(* IEC 61131-3 sources: Lasal/CPU_5344_V01/Class/MillPlane, 1 file *)

(* ---- MillPlane.st ---- *)
(*!
<Class
	Name               = "MillPlane"
	Revision           = "0.0"
	RealtimeTask       = "false"
	CyclicTask         = "false"
	BackgroundTask     = "false"
	Sigmatek           = "false"
	OSInterface        = "false"
	HighPriority       = "false"
	Automatic          = "false"
	UpdateMode         = "Prescan"
	SharedCommandTable = "true"
	Objectsize         = "(390,360)">
	<Channels>
		<Server Name="amount" Visualized="true" Initialize="false" WriteProtected="false" Retentive="false"/>
		<Server Name="ClassSvr" Visualized="false" Initialize="false" WriteProtected="true" Retentive="false"/>
		<Server Name="depth" Visualized="true" Initialize="false" WriteProtected="false" Retentive="false"/>
		<Server Name="feedRate" Visualized="true" Initialize="false" WriteProtected="false" Retentive="false"/>
		<Server Name="firsIdx" Visualized="true" Initialize="false" WriteProtected="false" Retentive="false"/>
		<Server Name="lowerRate" Visualized="true" Initialize="false" WriteProtected="false" Retentive="false"/>
		<Server Name="rnr" Visualized="true" Initialize="false" WriteProtected="false" Retentive="false"/>
		<Client Name="line1" Required="true" Internal="true"/>
		<Client Name="line2" Required="true" Internal="true"/>
		<Client Name="line3" Required="true" Internal="true"/>
		<Client Name="line4" Required="true" Internal="true"/>
		<Client Name="line5" Required="true" Internal="true"/>
		<Client Name="line6" Required="true" Internal="true"/>
	</Channels>
	<Network Name="MillPlane">
		<!-- List of Components in this network -->
		<Components>
			<Object
				Name       = "line1"
				Class      = "MillLine"
				Position   = "(150,120)"
				Visualized = "true">
				<Channels>
					<Server Name="ClassSvr"/>
					<Server Name="middleX"/>
					<Server Name="middleY"/>
					<Server Name="millType"/>
					<Server Name="radius"/>
					<Server Name="rnr"/>
					<Server Name="xGoal"/>
					<Server Name="yGoal"/>
				</Channels>
			</Object>
			<Object
				Name       = "line2"
				Class      = "MillLine"
				Position   = "(150,690)"
				Visualized = "true">
				<Channels>
					<Server Name="ClassSvr"/>
					<Server Name="middleX"/>
					<Server Name="middleY"/>
					<Server Name="millType"/>
					<Server Name="radius"/>
					<Server Name="rnr"/>
					<Server Name="xGoal"/>
					<Server Name="yGoal"/>
				</Channels>
			</Object>
			<Object
				Name       = "line3"
				Class      = "MillLine"
				Position   = "(720,120)"
				Visualized = "true">
				<Channels>
					<Server Name="ClassSvr"/>
					<Server Name="middleX"/>
					<Server Name="middleY"/>
					<Server Name="millType"/>
					<Server Name="radius"/>
					<Server Name="rnr"/>
					<Server Name="xGoal"/>
					<Server Name="yGoal"/>
				</Channels>
			</Object>
			<Object
				Name       = "line4"
				Class      = "MillLine"
				Position   = "(720,690)"
				Visualized = "true">
				<Channels>
					<Server Name="ClassSvr"/>
					<Server Name="middleX"/>
					<Server Name="middleY"/>
					<Server Name="millType"/>
					<Server Name="radius"/>
					<Server Name="rnr"/>
					<Server Name="xGoal"/>
					<Server Name="yGoal"/>
				</Channels>
			</Object>
			<Object
				Name       = "line5"
				Class      = "MillLine"
				Position   = "(1260,120)"
				Visualized = "true">
				<Channels>
					<Server Name="ClassSvr"/>
					<Server Name="middleX"/>
					<Server Name="middleY"/>
					<Server Name="millType"/>
					<Server Name="radius"/>
					<Server Name="rnr"/>
					<Server Name="xGoal"/>
					<Server Name="yGoal"/>
				</Channels>
			</Object>
			<Object
				Name       = "line6"
				Class      = "MillLine"
				Position   = "(1260,690)"
				Visualized = "true">
				<Channels>
					<Server Name="ClassSvr"/>
					<Server Name="middleX"/>
					<Server Name="middleY"/>
					<Server Name="millType"/>
					<Server Name="radius"/>
					<Server Name="rnr"/>
					<Server Name="xGoal"/>
					<Server Name="yGoal"/>
				</Channels>
			</Object>
		</Components>
		<Comments>
		</Comments>
		<!-- List of Connections in this network -->
		<Connections>
			<Connection Source="this.line1" Destination="line1.ClassSvr"/>
			<Connection Source="this.line2" Destination="line2.ClassSvr"/>
			<Connection Source="this.line4" Destination="line4.ClassSvr"/>
			<Connection Source="this.line3" Destination="line3.ClassSvr"/>
			<Connection Source="this.line5" Destination="line5.ClassSvr"/>
			<Connection Source="this.line6" Destination="line6.ClassSvr"/>
		</Connections>
		<!-- Headerfiles -->
		<Options>
		</Options>
	</Network>
</Class>
*)
MillPlane : CLASS
  //Servers:
	ClassSvr 	: SvrChCmd_DINT;
	rnr 	: SvrCh_DINT;
	depth 	: SvrCh_DINT;
	amount 	: SvrCh_DINT;
	feedRate 	: SvrCh_DINT;
	lowerRate 	: SvrCh_DINT;
	firsIdx 	: SvrCh_DINT;
  //Clients:
	line1 	: CltChCmd_MillLine;
	line2 	: CltChCmd_MillLine;
	line3 	: CltChCmd_MillLine;
	line4 	: CltChCmd_MillLine;
	line5 	: CltChCmd_MillLine;
	line6 	: CltChCmd_MillLine;
  //Variables:
		ptr 	: ^strMillPlane;
  //Functions:

	FUNCTION GLOBAL WritePtr
		VAR_INPUT
			iPtr 	: ^strMillPlane;
		END_VAR;

	FUNCTION WriteServers;

	FUNCTION VIRTUAL GLOBAL depth::Write
		VAR_INPUT
			input (EAX) 	: DINT;
		END_VAR
		VAR_OUTPUT
			result (EAX) 	: DINT;
		END_VAR;

	FUNCTION VIRTUAL GLOBAL amount::Write
		VAR_INPUT
			input (EAX) 	: DINT;
		END_VAR
		VAR_OUTPUT
			result (EAX) 	: DINT;
		END_VAR;

	FUNCTION VIRTUAL GLOBAL feedRate::Write
		VAR_INPUT
			input (EAX) 	: DINT;
		END_VAR
		VAR_OUTPUT
			result (EAX) 	: DINT;
		END_VAR;

	FUNCTION VIRTUAL GLOBAL lowerRate::Write
		VAR_INPUT
			input (EAX) 	: DINT;
		END_VAR
		VAR_OUTPUT
			result (EAX) 	: DINT;
		END_VAR;

	FUNCTION VIRTUAL GLOBAL firsIdx::Write
		VAR_INPUT
			input (EAX) 	: DINT;
		END_VAR
		VAR_OUTPUT
			result (EAX) 	: DINT;
		END_VAR;
  //Tables:
	FUNCTION @STD
		VAR_OUTPUT
			ret_code	: CONFSTATES;
		END_VAR;
	FUNCTION GLOBAL TAB @CT_;
END_CLASS;

#pragma using MillLine

FUNCTION VIRTUAL GLOBAL MillPlane::depth::Write
	VAR_INPUT
		input (EAX) 	: DINT;
	END_VAR
	VAR_OUTPUT
		result (EAX) 	: DINT;
	END_VAR

  if ptr <> NIL then
    depth := input;
    ptr^.depth := depth;
    result := depth;
  else
    result := ACCESS_DENIED;
  end_if;

END_FUNCTION

FUNCTION VIRTUAL GLOBAL MillPlane::amount::Write
	VAR_INPUT
		input (EAX) 	: DINT;
	END_VAR
	VAR_OUTPUT
		result (EAX) 	: DINT;
	END_VAR

  if ptr <> NIL then
    amount := input;
    ptr^.amount := amount;
    result := amount;
  else
    result := ACCESS_DENIED;
  end_if;

END_FUNCTION

FUNCTION VIRTUAL GLOBAL MillPlane::feedRate::Write
	VAR_INPUT
		input (EAX) 	: DINT;
	END_VAR
	VAR_OUTPUT
		result (EAX) 	: DINT;
	END_VAR

  if ptr <> NIL then
    feedRate := input;
    ptr^.feedRate := feedRate;
    result := feedRate;
  else
    result := ACCESS_DENIED;
  end_if;

END_FUNCTION

FUNCTION GLOBAL MillPlane::WritePtr
	VAR_INPUT
		iPtr 	: ^strMillPlane;
	END_VAR

  ptr := iPtr;
  WriteServers();
  firsIdx.Write(input:=0);

END_FUNCTION

FUNCTION MillPlane::WriteServers

  if ptr <> NIL then
    depth := ptr^.depth;
    amount := ptr^.amount;
    feedRate := ptr^.feedRate;
    lowerRate := ptr^.lowerRate;
  end_if;

END_FUNCTION

FUNCTION VIRTUAL GLOBAL MillPlane::lowerRate::Write
	VAR_INPUT
		input (EAX) 	: DINT;
	END_VAR
	VAR_OUTPUT
		result (EAX) 	: DINT;
	END_VAR

  if ptr <> NIL then
	  lowerRate := input;
    ptr^.lowerRate := lowerRate;
	  result := lowerRate;
  else
    result := ACCESS_DENIED;
  end_if;

END_FUNCTION

FUNCTION VIRTUAL GLOBAL MillPlane::firsIdx::Write
	VAR_INPUT
		input (EAX) 	: DINT;
	END_VAR
	VAR_OUTPUT
		result (EAX) 	: DINT;
	END_VAR

	firsIdx := input;
  if firsIdx >= 0 & firsIdx <= (cMaxMillLinesInPlane-2) & ptr<>NIL then
    line1.WritePtr(iPtr:=#ptr^.lines[firsIdx]);
    line2.WritePtr(iPtr:=#ptr^.lines[firsIdx+1]);
//    line3.WritePtr(iPtr:=#ptr^.lines[firsIdx+2]);
//    line4.WritePtr(iPtr:=#ptr^.lines[firsIdx+3]);
//    line5.WritePtr(iPtr:=#ptr^.lines[firsIdx+4]);
//    line6.WritePtr(iPtr:=#ptr^.lines[firsIdx+5]);
    line1.rnr.Write(input:=firsIdx+1);
    line2.rnr.Write(input:=firsIdx+2);
//    line3.rnr.Write(input:=firsIdx+3);
//    line4.rnr.Write(input:=firsIdx+4);
//    line5.rnr.Write(input:=firsIdx+5);
//    line6.rnr.Write(input:=firsIdx+6);
  else
    result:=ACCESS_DENIED;
    firsIdx-=1;
  end_if;
	result := firsIdx;

END_FUNCTION
